// Brief: Master Arm Master Slave Control
FUNCTION_BLOCK PUBLIC FB_StateCtrlInit EXTENDS FB_SlaveArmCtrlBase
VAR_INPUT
END_VAR
VAR_OUTPUT
END_VAR
VAR
	m_initState :INT :=0;
END_VAR

METHOD PUBLIC init : BOOL
VAR_IN_OUT CONSTANT
	i_slaveArm	:FB_SlaveArm;
END_VAR
VAR_IN_OUT 
	r_slaveArmCtrlCmd :ST_SlaveArmCtrlCmds;
END_VAR

VAR
	i:INT;
END_VAR
SUPER^.Init(i_slaveArm,r_slaveArmCtrlCmd);
m_jntEnableFlag:=g_zeroVec8i;
END_METHOD

END_FUNCTION_BLOCK

(* stored: Version 1.1.0.1, ProductVersion 3.1.4024.12
   POU FB_StateCtrlInit: Id {2f1b91d8-ebd5-4b63-92d8-450fe3a94973}, SpecialFunc None
   Method init: Id {0eca198b-2030-4cc0-a250-a6bdc9d0e230} *)
